Staubli VAL3: monitorAreaEn.pjx

--- monitorAreaEn.pjx ---
Parameters version=s7.9.1 stackSize=5000 millimeterUnit=true
Program file=checkCube.pgx
Program file=checkCylinder.pgx
Program file=checkFrame.pgx
Program file=checkSphere.pgx
Program file=createCube.pgx
Program file=createCylinder.pgx
Program file=createFrame.pgx
Program file=createSphere.pgx
Program file=example.pgx
Program file=init.pgx
Program file=readme.pgx
Program file=start.pgx
Program file=stop.pgx
Data file=monitorAreaEn.dtx
Library alias=io path=Disk://io/io.pjx

--- monitorAreaEn.dtx ---
public num nDistXCube[10]
public num nDistYCube[10]
public num nDistZCube[10]
public num nDistZCylinder[10]
public num nNumberCube = 9
public num nNumberCylinder = 9
public num nNumberFrame
public num nNumberSphere = 9
public num nRadiusCylinder[10]
public num nRadiusSphere[10]
  [9] = 600
public bool bCreateCube[10]
public bool bCreateCylinder[10]
bool bCreateFrame[10]
public bool bCreateSphere[10]
  [9] = true
frame fCube[10]
  [0] = {fatherId=world[0]}
  [1] = {fatherId=world[0]}
  [2] = {fatherId=world[0]}
  [3] = {fatherId=world[0]}
  [4] = {fatherId=world[0]}
  [5] = {fatherId=world[0]}
  [6] = {fatherId=world[0]}
  [7] = {fatherId=world[0]}
  [8] = {fatherId=world[0]}
  [9] = {fatherId=world[0]}
frame fCylinder[10]
  [0] = {fatherId=world[0]}
  [1] = {fatherId=world[0]}
  [2] = {fatherId=world[0]}
  [3] = {fatherId=world[0]}
  [4] = {fatherId=world[0]}
  [5] = {fatherId=world[0]}
  [6] = {fatherId=world[0]}
  [7] = {fatherId=world[0]}
  [8] = {fatherId=world[0]}
  [9] = {fatherId=world[0]}
frame fFrameZone[10]
  [0] = {fatherId=world[0]}
  [1] = {fatherId=world[0]}
  [2] = {fatherId=world[0]}
  [3] = {fatherId=world[0]}
  [4] = {fatherId=world[0]}
  [5] = {fatherId=world[0]}
  [6] = {fatherId=world[0]}
  [7] = {fatherId=world[0]}
  [8] = {fatherId=world[0]}
  [9] = {fatherId=world[0]}
frame fTableExample = {z=-50, fatherId=world[0]}
public pointRx pOriginCube[10]
  [0] = {fatherId=world[0]}
  [1] = {fatherId=world[0]}
  [2] = {fatherId=world[0]}
  [3] = {fatherId=world[0]}
  [4] = {fatherId=world[0]}
  [5] = {fatherId=world[0]}
  [6] = {fatherId=world[0]}
  [7] = {fatherId=world[0]}
  [8] = {fatherId=world[0]}
  [9] = {fatherId=world[0]}
public pointRx pOriginCylinder[10]
  [0] = {fatherId=world[0]}
  [1] = {fatherId=world[0]}
  [2] = {fatherId=world[0]}
  [3] = {fatherId=world[0]}
  [4] = {fatherId=world[0]}
  [5] = {fatherId=world[0]}
  [6] = {fatherId=world[0]}
  [7] = {fatherId=world[0]}
  [8] = {fatherId=world[0]}
  [9] = {fatherId=world[0]}
public pointRx pOriginSphere[10]
  [0] = {fatherId=world[0]}
  [1] = {fatherId=world[0]}
  [2] = {fatherId=world[0]}
  [3] = {fatherId=world[0]}
  [4] = {fatherId=world[0]}
  [5] = {fatherId=world[0]}
  [6] = {fatherId=world[0]}
  [7] = {fatherId=world[0]}
  [8] = {fatherId=world[0]}
  [9] = {y=300, z=1200, rx=180, fatherId=world[0]}
pointRx pStartExample = {x=400, z=100, fatherId=world[0]}
pointRx pStartExample2 = {x=600, z=-50, fatherId=world[0]}

--- start.pgx ---
program start()
begin
  call example()
end

--- checkCube.pgx ---
public program checkCube(tool x_tTool, num x_nCube, bool& x_bCheckCube[], bool& x_bError[])
  local bool l_bPositive
  local bool l_bNegative
  local point l_pPointHere
begin
  //Header begin
  //Description of program
  //  This program checks if the tool is inside the specified cubic area
  //
  //Input parameters
  //  tool x_tTool :
  //    role : defines the tool that you want to monitor the position of
  //  num x_nCube :
  //    role : number of the cubic zone to be monitored (in order of creation)
  //    possible values : number of an existing cubic zone
  //
  //Output parameters
  //  bool x_bCheckCube :
  //    role : set to true if the tool is inside the cubic zone and false otherwise
  //  bool x_bError :
  //    role : set to true if the cubic zone does not exist and false otherwise
  //
  //Example :
  //  call checkCube(tTool, 1, bOK, bErr)
  //
  //History
  //  Creation : 16-04-08 - f.Rob
  //  updated for SLAC KN
  //Header end

  //Test if the cube that you want to monitor is created
  call init()
  //DEBUG:putln("pgm MON: checkCube()")
  if x_nCube>nNumberCube
    x_bError=true
    stopMove()
    disablePower()
    //User interface
    popUpMsg("Cube Zone #"+toString("",x_nCube)+" has not been created."+chr(10)+"Stop the program !!!")
    delay(3)
    return
  endIf
  x_bError=false
  x_bCheckCube=false
  if bCreateCube[x_nCube]
    l_pPointHere=here(x_tTool,fCube[x_nCube])
    //Check if the tool is inside area just on Z component
    if l_pPointHere.trsf.z>0 and l_pPointHere.trsf.z<nDistZCube[x_nCube]
      //Check if positive or negative of Y
      l_bPositive=l_pPointHere.trsf.y>0 and l_pPointHere.trsf.y<nDistYCube[x_nCube] and nDistYCube[x_nCube]>0
      l_bNegative=l_pPointHere.trsf.y<0 and l_pPointHere.trsf.y>nDistYCube[x_nCube] and nDistYCube[x_nCube]<0
      if l_bPositive or l_bNegative
        //Check if positive or negative of X
        l_bPositive=l_pPointHere.trsf.x>0 and l_pPointHere.trsf.x<nDistXCube[x_nCube] and nDistXCube[x_nCube]>0
        l_bNegative=l_pPointHere.trsf.x<0 and l_pPointHere.trsf.x>nDistXCube[x_nCube] and nDistXCube[x_nCube]<0
        //Test if the tool is inside the cube
        if l_bPositive or l_bNegative
          x_bCheckCube=true
        endIf
      endIf
    endIf
  endIf
end

--- checkCylinder.pgx ---
public program checkCylinder(tool x_tTool, num x_nCylinder, bool& x_bCheckCylind[], bool& x_bError[])
  local point l_pPointHere
  local point l_pNewOrigin
begin
  //Header begin
  //Description of program
  //  This program checks if the tool is inside the specified cylindrical zone
  //
  //Input parameters
  //  point x_tTool :
  //    role : defines the tool that you want to monitor the position of
  //  num x_nCylinder :
  //    role : number of the cylindrical zone to be monitored (in order of creation)
  //    possible values :  number of an existing cylindrical zone
  //
  //Output parameters
  //  num x_bCheckCylind :
  //    role : set to true if the tool is inside the cylindrical zone and false otherwise
  //  bool x_bError :
  //    role : set to true if the cylindrical zone does not exist and false otherwise
  //
  //Example
  //  call checkCylinder(flange,5,bOK,bErr)
  //
  //History
  //  Creation : 16-04-08 - f.Rob
  //  updated for SLAC KN
  //Header end

  //Test if the cylinder that you want to monitor is created
  call init()
  //DEBUG:putln("pgm MON: checkCylinder()")
  if x_nCylinder>nNumberCylinder
    x_bError=true
    stopMove()
    disablePower()
    //User interface
    popUpMsg("Cylinder Zone #"+toString("",x_nCylinder)+" has not been created."+chr(10)+"Stop the program !!!")
    delay(3)
    return
  endIf
  x_bError=false
  x_bCheckCylind=false
  if bCreateCylinder[x_nCylinder]
    //here() returns the current position of x_tTool tool in fCylinder frame.
    l_pPointHere=here(x_tTool,fCylinder[x_nCylinder])
    //Check if inside
    if l_pPointHere.trsf.z>=0 and l_pPointHere.trsf.z<=nDistZCylinder[x_nCylinder]
      //Inside the cylinder
      l_pNewOrigin=compose(pOriginCylinder[x_nCylinder],world,{0,0,l_pPointHere.trsf.z,0,0,0})
      //Test if the tool is inside the cylinder
      if distance(l_pNewOrigin,l_pPointHere)<=nRadiusCylinder[x_nCylinder]
        x_bCheckCylind=true
      endIf
    endIf
  endIf
end

--- checkFrame.pgx ---
public program checkFrame(tool x_tTool, num x_nFrame, bool& x_bCheckFrame[], bool& x_bError[])
  local point l_pPointHere
begin
  //Header begin
  //Description of program
  //  Monitors Z position of a tool center point in regards to a frame.
  //  It will set to "true" a bool variable when Z<0 and set to "false" otherwise
  //
  //Input parameters
  //  point x_tTool :
  //    role : defines the tool that you want to monitor the position of
  //  num x_nFrame :
  //    role : number of the frame zone to be monitored (in order of creation)
  //    possible values : number of an existing frame zone
  //
  //Output parameters
  //  num x_bCheckFrame :
  //    role : set to true if the Z tool is above the frame and set to false otherwise
  //  bool x_bError :
  //    role : set to true if the frame zone does not exist and false otherwise
  //
  //Example
  //  call checkFrame(flange,3,bOK,bErr)
  //
  //History
  //  Creation : 16-04-08 - f.Rob
  //Header end

  //Test if the frame that you want to monitor is created
  if x_nFrame>nNumberFrame
    x_bError=true
    stopMove()
    disablePower()
    //User interface
   popUpMsg("Frame area number "+toString("",x_nFrame)+" has not been created."+chr(10)+"Stop the program !!!")
   delay(3)
   return
  endIf
  x_bError=false
  x_bCheckFrame=false
  if bCreateFrame[x_nFrame-1]
    //here() returns the current position of x_tTool tool in x_fFrame frame.
    l_pPointHere=here(x_tTool,fFrameZone[x_nFrame-1])
    //Test if the tool is above the frame
    if l_pPointHere.trsf.z>0
       x_bCheckFrame=true
    endIf
  endIf
end

--- checkSphere.pgx ---
public program checkSphere(tool x_tTool, num x_nSphere, bool& x_bCheckSphere[], bool& x_bError[])
  local point l_pPointHere
  local num l_nIndex
begin
  //Header begin
  //Description of program
  //  This program checks if the tool is inside the spherical zone
  //
  //Input parameters
  //  point x_tTool :
  //    role : defines the tool that you want to monitor the position of
  //  num x_nSphere :
  //    role : number of the spherical zone to be monitored (in order of creation)
  //    possible values : number of an existing spherical zone
  //
  //Output parameters
  //  num x_bCheckSphere :
  //    role : set to true if the tool is inside the spherical zone and false otherwise
  //  bool x_bError :
  //    role : set to true if the frame zone does not exist and false otherwise
  //
  //Example
  //  call checkSphere(flange,1,bOK,bErr)
  //
  //History
  //  Creation : 16-04-08 - f.Rob
  //  updated for SLAC KN
  //Header end

  //Test if the sphere that you want to monitor is created
  call init()
  //DEBUG:putln("pgm MON:checkSphere()")
  if x_nSphere>nNumberSphere
    x_bError=true
    stopMove()
    disablePower()
    //User interface
    popUpMsg("Sphere Zone #"+toString("",x_nSphere)+" has not been created."+chr(10)+"Stop the program !!!")
    delay(3)
    return
  endIf
  x_bError=false
  x_bCheckSphere=false
  if bCreateSphere[x_nSphere]
    //here() returns the current position of x_tTool tool in world frame.
    l_pPointHere=here(x_tTool,world)
    //Check if inside specified sphere
    if distance(pOriginSphere[x_nSphere],l_pPointHere)<nRadiusSphere[x_nSphere]
      x_bCheckSphere=true
    endIf
  endIf
end

--- createCube.pgx ---
public program createCube(point x_pOrigin, num x_nDistanceX, num x_nDistanceY, num x_nDistanceZ, bool& x_bError[])
  local trsf l_trsfCopy
  local point l_pOrigine
  local num l_nSizeTab
begin
  //Header begin
  //Description of program
  //  This program creates a cubic area
  //  defined by a point and 3 distances X, Y, Z
  //
  //  KN note:  cube is considered 'active' if bCreateCube = true.  This boolean is cleared in pgm mnuTeachCube().
  //
  //Input parameters
  //  point x_pOrigin :
  //    role : defines the origin of the cube
  //  num x_nDistanceX :
  //    role : defines the dimension about the world's X axis
  //  num x_nDistanceY :
  //    role : defines the dimension about the world's Y axis
  //  num x_nDistanceZ :
  //    role : defines the dimension about the world's Z axis
  //
  //Output parameters
  //  bool x bError :
  //    role : set to true when the cubic area could not be created, false otherwise
  //
  //Example
  //  call createCube(pOriginCube,400, 200, 100,bOK)
  //
  //History
  //  Creation : 16-04-08 - f.Rob
  //  Initial release KN
  //
  //Header end

  //Find the smallest array, this will define the maximum number of zones that can created
  l_nSizeTab=size(pOriginCube)
  if size(fCube)<l_nSizeTab
    l_nSizeTab=size(fCube)
  endIf
  if size(nDistXCube)<l_nSizeTab
    l_nSizeTab=size(nDistXCube)
  endIf
  if size(nDistYCube)<l_nSizeTab
    l_nSizeTab=size(nDistYCube)
  endIf
  if size(nDistZCube)<l_nSizeTab
    l_nSizeTab=size(nDistZCube)
  endIf
  //Test if it's possible to creates a new cube (not exceed the maximum size of the smallest array)
  if (nNumberCube>l_nSizeTab-1)
    x_bError=true
    popUpMsg("Cube area number "+toString("",nNumberCube)+" cannot be created : you can create only "+toString("",l_nSizeTab)+" (0.."+toString("",l_nSizeTab-1)+") area of this type")
    return
  endIf
  //Build the cube
  pOriginCube[nNumberCube].trsf=position(x_pOrigin,world)
  if setFrame(pOriginCube[nNumberCube],compose(pOriginCube[nNumberCube],world,{x_nDistanceX,0,0,0,0,0}),compose(pOriginCube[nNumberCube],world,{0,x_nDistanceY,0,0,0,0}),fCube[nNumberCube])==0
     bCreateCube[nNumberCube]=true
  endIf
  //Distances x y z
  nDistXCube[nNumberCube]=x_nDistanceX
  nDistYCube[nNumberCube]=x_nDistanceY
  nDistZCube[nNumberCube]=x_nDistanceZ
  //Regolate the frame
  l_trsfCopy=fCube[nNumberCube].trsf
  fCube[nNumberCube].trsf={l_trsfCopy.x,l_trsfCopy.y,l_trsfCopy.z,0,0,0}

  nNumberCube=nNumberCube+1
end

--- createCylinder.pgx ---
public program createCylinder(point x_pOrigin, num x_nRadius, num x_nDistanceZ, bool& x_bError[])
  local num l_nSizeTab
begin
  //Header begin
  //Description of program
  //  This program creates a cylindrical area
  //  defined by a point,a Radius and a Distance
  //
  // KN note:  cylinder considered 'active' if bCreateCylinder==true.  This boolean is cleared in pgm mnuTeachCyl()
  //
  //Input parameters
  //  point x_pOrigin :
  //    role : defines the origin and the diameter of the cylinder
  //  num x_nRadius :
  //    role : defines the radius of the cylinder
  //  num x_nDistanceZ :
  //    role : defines the height of the cylinder about Z world
  //
  //Output parameters
  //  bool x bError :
  //    role : set to true when the cylinder area could not be created, false otherwise
  //
  //Example
  //  call createCylinder(pCenterCylinder,100,350,bOK)
  //
  //History
  //  Creation : 16-04-08 - f.Rob
  //Header end

  //Find the smallest array, this will define the maximum number of zones that can created
  l_nSizeTab=size(pOriginCylinder)
  if size(fCylinder)<l_nSizeTab
    l_nSizeTab=size(fCylinder)
  endIf
  if size(nRadiusCylinder)<l_nSizeTab
    l_nSizeTab=size(nRadiusCylinder)
  endIf
  if size(nDistZCylinder)<l_nSizeTab
    l_nSizeTab=size(nDistZCylinder)
  endIf
  //Test if it's possible to creates a new cylinder (not exceed the maximum size of the smallest array)
  if (nNumberCylinder>l_nSizeTab-1)
    x_bError=true
    popUpMsg("Cylinder area number "+toString("",nNumberCylinder)+" cannot be created : you can create only "+toString("",l_nSizeTab)+" (0.."+toString("",l_nSizeTab-1)+") area of this type")
    return
  endIf
  //Build the cylinder
  pOriginCylinder[nNumberCylinder].trsf=position(x_pOrigin,world)
  if setFrame(pOriginCylinder[nNumberCylinder],compose(pOriginCylinder[nNumberCylinder],world,{x_nRadius,0,0,0,0,0}),compose(pOriginCylinder[nNumberCylinder],world,{0,x_nRadius,0,0,0,0}),fCylinder[nNumberCylinder])==0
    bCreateCylinder[nNumberCylinder]=true
  endIf
  //Copy all parameters
  nRadiusCylinder[nNumberCylinder]=x_nRadius
  nDistZCylinder[nNumberCylinder]=x_nDistanceZ

  nNumberCylinder=nNumberCylinder+1
end

--- createFrame.pgx ---
public program createFrame(frame x_fFrame, bool& x_bError[])
  local num l_nSizeTab
begin
  //Header begin
  //Description of program
  //  This program creates an area for monitoring the Z position of
  //  a tool center point in regards to a frame.
  //
  //Input parameters
  //  frame x_fFrame :
  //    role : defines the frame that you want to use for monitoring the z value
  //
  //Output parameters
  //  bool x bError :
  //    role : set to true when the frame area could not be created, false otherwise
  //
  //Example
  //  call createFrame(fTable,bOK)
  //
  //History
  //  Creation : 16-04-08 - f.Rob
  //Header end


  l_nSizeTab=size(fFrameZone)

  //Test if it's possible to creates a new cylinder (not exceed the maximum size of the array)
  if (nNumberFrame>l_nSizeTab-1)
    x_bError=true
    popUpMsg("Frame area number "+toString("",nNumberFrame)+" cannot be created : you can create only "+toString("",l_nSizeTab)+" (0.."+toString("",l_nSizeTab-1)+") area of this type")
    return
  endIf
  //Build the frame
  fFrameZone[nNumberFrame]=x_fFrame
  bCreateFrame[nNumberFrame]=true

  nNumberFrame=nNumberFrame+1
end

--- createSphere.pgx ---
public program createSphere(point x_pOrigin, num x_nRadius, bool& x_bError[])
  local num l_nIndex
  local num l_nSizeTab
begin
  //Header begin
  //Description of program
  //  This program creates a spherical area
  //  defined by a point and a distance
  //
  //  KN note:  sphere is considered 'active' if bCreateSphere==true.  This bool is cleared in pgm mnuTeachSphere().
  //
  //Input parameters
  //  point x_pOrigin :
  //    role : defines the center of the zone that you want to create
  //  num x_nRadius :
  //    role : defines the radius of the sphere
  //
  //Example
  //  call createSphere(pCenterSphere,350,bOK)
  //
  //History
  //  Creation : 16-04-08 - f.Rob
  //Header end

  //Find the smallest array, this will define the maximum number of zones that can created
  l_nSizeTab=size(pOriginSphere)
  if (size(nRadiusSphere)<l_nSizeTab)
    l_nSizeTab=size(nRadiusSphere)
  endIf
  //Test if it's possible to creates a new sphere (not exceed the maximum size of the smallest array)
  if (nNumberSphere>l_nSizeTab-1)
    x_bError=true
    popUpMsg("Sphere area number "+toString("",nNumberSphere)+" cannot be created : you can create only "+toString("",l_nSizeTab)+" (0.."+toString("",l_nSizeTab-1)+") area of this type")
    return
  endIf
  //Build te sphere
  pOriginSphere[nNumberSphere].trsf=position(x_pOrigin,world)
  nRadiusSphere[nNumberSphere]=x_nRadius
  bCreateSphere[nNumberSphere]=true

  nNumberSphere=nNumberSphere+1
end

--- example.pgx ---
program example()
  local num l_nDistXCube
  local num l_nDistYCube
  local num l_nDistZCube
  local bool l_bSecuCube
  local bool l_bSecuFrame
  local bool l_bSecuSphere
  local bool l_bSecuCylinder
  local bool l_bSecuSphere2
  local bool l_bErrCube
  local bool l_bErrFrame
  local bool l_bErrSphere
  local bool l_bErrSphere2
  local bool l_bErrCylinder
begin
  //Header begin
  //Description of programm
  //  This is an example for use this library.
  //  In this example 2 spherical,1 frame area,
  //  1 cubic area, 1 cylindrical area are monitoring
  //
  //History
  //  Creation : 16-04-08 - f.Rob
  //Header end

  call init()
  //Creation of areas
  call createFrame(fTableExample,l_bErrFrame)
  call createCube(pStartExample,200 ,200 ,200,l_bErrCube)
  call createSphere(pStartExample,500,l_bErrSphere)
  call createSphere(pStartExample2,400,l_bErrSphere2)
  call createCylinder(pStartExample, 200, 600,l_bErrCylinder)
  if l_bErrFrame or l_bErrCube or l_bErrSphere or l_bErrSphere2 or l_bErrCylinder
    //Error on one of the creation
  else
    userPage()
    cls()
    while true
      //Areas monitoring
      call checkCube(flange,1,l_bSecuCube,l_bErrFrame)
      call checkFrame(flange,1,l_bSecuFrame,l_bErrCube)
      call checkSphere(flange,1,l_bSecuSphere,l_bErrSphere)
      call checkSphere(flange,2,l_bSecuSphere2,l_bErrSphere2)
      call checkCylinder(flange,1,l_bSecuCylinder,l_bErrCylinder)
      if l_bErrFrame or l_bErrCube or l_bErrSphere or l_bErrSphere2 or l_bErrCylinder
        //Error on one of the checks
      else
        if !l_bSecuCube
          putln("Tool is outside CUBE")
        endIf
        if !l_bSecuFrame
          putln("Tool is outside FRAME")
        endIf
        if !l_bSecuSphere
          putln("Tool is outside SPHERE")
        endIf
        if !l_bSecuSphere2
          putln("Tool is outside SPHERE 2")
        endIf
        if !l_bSecuCylinder
          putln("Tool is outside CYLINDER")
        endIf
        if l_bSecuCube and l_bSecuFrame and l_bSecuSphere and l_bSecuCylinder and l_bSecuSphere2
          putln("OK tool")
        endIf
        delay(0)
        cls()
      endIf
    endWhile
  endIf
end

--- init.pgx ---
public program init()
begin
  //Header begin
  //Description of program
  //  This program initializes the library's global variables.
  //  It has to be called once at the beginning of the users program
  //
  //History
  //  Creation : 16-04-08 - f.Rob
  //  KN: set quantity = 9 = max index of arrays (0-9)
  //Header end

  nNumberCylinder=nNumberCube=nNumberSphere=nNumberFrame=9
end

--- readme.pgx ---
program readme()
begin
  //Title: Monitoring the robot position in regards to an area
  //
  //General description :
  //
  //  Possibility to monitor the current Z position  value compared to a frame
  //  Possibility to monitor a distance to a point (spherical zone)
  //  Possibility to monitor the current position of a tool in a Cube
  //  Possibility to monitor the current position of a tool in a Cylinder
  //  Possibility to monitor up to 40 areas (10 identical areas per solid)
  //  (example : 10 spherical areas and 10 cubic areas)
  //
  //Hardware required :
  //  - Robot system    : any Staubli robot
  //  - Peripherals     : no peripherals required
  //
  //VAL3 options :
  //  - VAL3 version    : 6.4
  //  - VAL3 licenses   : no licenses required
  //  - VAL3 add-ons    : none
  //
  //Library version     : 6.4.1.0
  //
  //Public variables    : none
  //
  //Included libraries  : none
  //
  //Miscellaneous       : ---
  //
  //Keywords            : monitor, controle, position, area, zone, cube, cylinder, cylindre, sphere, frame, plan


end

--- stop.pgx ---
program stop()
begin
  popUpMsg("Pending movement commands have been canceled")
  resetMotion()
end
